// TwinCAT 3 PLC project ServoMotion_Library
// Title: ServoMotion_Lib
// Company: Chua Siang Poh
// Author: Chua Siang Poh
// ProjectVersion: 1.0
// Description: For projects that require at least 1 motion axis. The library is meant as an easy-to-setup module. Only requring the change of a parameter. Other motion functions are exposed as a method. Includes a very simple/crude type of linear interpolation.
// ProgramVersion: 3.1.0.8
// libraries:
//   Tc2_MC2, * (Beckhoff Automation GmbH)
//   Tc2_Standard, * (Beckhoff Automation GmbH)
//   Tc2_System, * (Beckhoff Automation GmbH)
//   Tc3_Interfaces, * (Beckhoff Automation GmbH)
//   Tc3_Module, * (Beckhoff Automation GmbH)
// project tree:
//   Custom Datatypes/ Motion_Axis.TcDUT, Motion_AxisGroup.TcDUT, Motion_HmiToPlc.TcDUT, Motion_PlcToHmi.TcDUT, ServoMotion_FunctionResult.TcDUT
//   GVL/ ServoMotion_GVL.TcGVL
//   / Interpolate.TcPOU, Servo.TcPOU, ServoMotion_Parameters.TcGVL
//   Version/ Global_Version.TcGVL
// (motion and I/O tree: see PLC project serialcommunication)
// real-time tasks:
//   TASK PlcTask: cycle T#10ms, priority 20, ADS port 350

// ---- Custom Datatypes/Motion_Axis.TcDUT
TYPE Motion_Axis :
STRUCT
	AXIS 					: AXIS_REF;
	HOME_CALIBRATION AT %I* : BOOL;
END_STRUCT
END_TYPE

// ---- Custom Datatypes/Motion_AxisGroup.TcDUT
TYPE Motion_AxisGroup :
STRUCT
	V_X			: LREAL;
	V_Y			: LREAL;
	X_AXIS		: INT;
	Y_AXIS		: INT;
	STATE		: INT;
	Y_IS_MASTER	: BOOL;
	X_DONE		: BOOL;
	Y_DONE		: BOOL;
END_STRUCT
END_TYPE

// ---- Custom Datatypes/Motion_HmiToPlc.TcDUT
TYPE Motion_HmiToPlc :
STRUCT
	TARGET_POSITION 	: LREAL;
	TARGET_VELOCITY 	: LREAL;
	TARGET_ACCELERATION : LREAL;
	TARGET_DECELERATION	: LREAL;
	TARGET_JERK			: LREAL;
	CONTROLLER_OVERRIDE	: LREAL;
	SERVO_ON			: BOOL;
	SERVO_ON_FW			: BOOL;
	SERVO_ON_BW			: BOOL;
	SERVO_OFF			: BOOL;
	SERVO_MOVE_ABS		: BOOL;
	SERVO_MOVE_REL		: BOOL;
	SERVO_HOME			: BOOL;
	SERVO_RESET			: BOOL;
	SERVO_JOG_MODE		: BOOL := FALSE;
	SERVO_JOG_FW_FAST	: BOOL;
	SERVO_JOG_BW_FAST	: BOOL;
	SERVO_JOG_FW_SLOW	: BOOL;
	SERVO_JOG_BW_SLOW	: BOOL;
END_STRUCT
END_TYPE

// ---- Custom Datatypes/Motion_PlcToHmi.TcDUT
TYPE Motion_PlcToHmi :
STRUCT
	actPos				: LREAL;
	actVelo				: LREAL;
	setPos				: LREAL; 
	setVelo 			: LREAL; 
	controller_override : LREAL;
	ErrorID				: UDINT;
	hasError			: BOOL;
	isDisabled 			: BOOL;
	isFwDisabled 		: BOOL;
	isBwDisabled 		: BOOL;
	isCalibrated		: BOOL;
	hasJob				: BOOL;
	isNotMoving 		: BOOL;
	isPositiveDirection : BOOL;
	isNegativeDirection : BOOL;            
    isInTarget 			: BOOL;            
    isInRange 			: BOOL;              
END_STRUCT
END_TYPE

// ---- Custom Datatypes/ServoMotion_FunctionResult.TcDUT
TYPE ServoMotion_FunctionResult :
(
	MOTION_OK := -1,
	MOTION_BUSY := 0,
	MOTION_UNKNOWN_AXIS,
	MOTION_UNKNOWN_AXIS_GROUP,
	MOTION_UNKNOWN_SAME_AXIS_IN_GROUP,
	MOTION_COMMAND_ABORTED,
	MOTION_ERROR
);
END_TYPE

// ---- GVL/ServoMotion_GVL.TcGVL
VAR_GLOBAL
	HmiToPlc	: ARRAY[1..MAX_AXES] OF Motion_HmiToPlc;
	PlcToHmi	: ARRAY[1..MAX_AXES] OF Motion_PlcToHmi;
	AXIS		: ARRAY[1..MAX_AXES] OF Motion_Axis;
END_VAR

// ---- ServoMotion_Parameters.TcGVL
VAR_GLOBAL CONSTANT
	MAX_AXES 		: INT := 2;
	MAX_AXIS_GROUPS	: INT := 1;
END_VAR

// ---- Version/Global_Version.TcGVL
// This function has been automatically generated from the project information.
VAR_GLOBAL CONSTANT
	{attribute 'const_non_replaced'}
	stLibVersion_ServoMotion_Lib : ST_LibVersion := (iMajor := 1, iMinor := 0, iBuild := 0, iRevision := 0, sVersion := '1.0');
END_VAR

// ---- Interpolate.TcPOU
FUNCTION_BLOCK Interpolate EXTENDS Servo
VAR_INPUT
END_VAR
VAR_OUTPUT
END_VAR
VAR
	fbGearIn 	: ARRAY [1..MAX_AXIS_GROUPS] OF MC_GEARIN;
	fbGearOut 	: ARRAY [1..MAX_AXIS_GROUPS] OF MC_GEAROUT;
	AXISGROUP	: ARRAY [1..MAX_AXIS_GROUPS] OF Motion_AxisGroup;
END_VAR

;

METHOD PUBLIC Set_AxisGroup : ServoMotion_FunctionResult
VAR_INPUT
	AXIS_GROUP_INDEX	: INT;
	X_AXIS_INDEX		: INT;
	Y_AXIS_INDEX		: INT;
END_VAR
IF AXIS_GROUP_INDEX < 1 OR AXIS_GROUP_INDEX > MAX_AXIS_GROUPS THEN
	Set_AxisGroup := ServoMotion_FunctionResult.MOTION_UNKNOWN_AXIS_GROUP;
ELSIF X_AXIS_INDEX < 1 OR X_AXIS_INDEX > MAX_AXES THEN
	Set_AxisGroup := ServoMotion_FunctionResult.MOTION_UNKNOWN_AXIS;
ELSIF Y_AXIS_INDEX < 1 OR Y_AXIS_INDEX > MAX_AXES THEN
	Set_AxisGroup := ServoMotion_FunctionResult.MOTION_UNKNOWN_AXIS;
ELSIF X_AXIS_INDEX = Y_AXIS_INDEX THEN
	Set_AxisGroup := ServoMotion_FunctionResult.MOTION_UNKNOWN_SAME_AXIS_IN_GROUP;
ELSE
	AXISGROUP[AXIS_GROUP_INDEX].X_AXIS := X_AXIS_INDEX;
	AXISGROUP[AXIS_GROUP_INDEX].Y_AXIS := Y_AXIS_INDEX;
	AXISGROUP[AXIS_GROUP_INDEX].STATE := -10;
	Set_AxisGroup := ServoMotion_FunctionResult.MOTION_OK;
END_IF
END_METHOD

METHOD PROTECTED Servo_GearIn : ServoMotion_FunctionResult
VAR_INPUT
	GROUP		: INT;
	MASTER		: INT;
	SLAVE		: INT;
	RATIO		: LREAL;
END_VAR
IF GROUP < 1 OR GROUP > MAX_AXIS_GROUPS THEN
	Servo_GearIn := ServoMotion_FunctionResult.MOTION_UNKNOWN_AXIS_GROUP;
ELSIF MASTER < 1 OR MASTER > MAX_AXES THEN
	Servo_GearIn := ServoMotion_FunctionResult.MOTION_UNKNOWN_AXIS;
ELSIF SLAVE < 1 OR SLAVE > MAX_AXES THEN
	Servo_GearIn := ServoMotion_FunctionResult.MOTION_UNKNOWN_AXIS;
ELSIF MASTER = SLAVE THEN
	Servo_GearIn := ServoMotion_FunctionResult.MOTION_UNKNOWN_SAME_AXIS_IN_GROUP;
ELSE
	fbGearIn[GROUP](
		Master:= AXIS[MASTER].AXIS, 
		Slave:= AXIS[SLAVE].AXIS, 
		Execute:= TRUE, 
		RatioNumerator:= RATIO, 
		RatioDenominator:= 1 );
	IF fbGearIn[GROUP].InGear THEN
		fbGearIn[GROUP](
			Master:= AXIS[MASTER].AXIS, 
			Slave:= AXIS[SLAVE].AXIS, 
			Execute:= FALSE );
		Servo_GearIn := ServoMotion_FunctionResult.MOTION_OK;
	ELSIF fbGearIn[GROUP].Error THEN
		fbGearIn[GROUP](
			Master:= AXIS[MASTER].AXIS, 
			Slave:= AXIS[SLAVE].AXIS, 
			Execute:= FALSE );
		Servo_GearIn := ServoMotion_FunctionResult.MOTION_ERROR;
	ELSIF fbGearIn[GROUP].CommandAborted THEN 
		fbGearIn[GROUP](
			Master:= AXIS[MASTER].AXIS, 
			Slave:= AXIS[SLAVE].AXIS, 
			Execute:= FALSE );
		Servo_GearIn := ServoMotion_FunctionResult.MOTION_COMMAND_ABORTED; 
	ELSE
		Servo_GearIn:= ServoMotion_FunctionResult.MOTION_BUSY;
	END_IF
END_IF
END_METHOD

METHOD PROTECTED Interpolate : ServoMotion_FunctionResult
VAR_INPUT
	GROUP			: INT;
	TO_X_POSITION	: LREAL;
	TO_Y_POSITION	: LREAL;
	VELOCITY		: LREAL;
END_VAR
VAR
	delta_t : LREAL;
	delta_x : LREAL;
	delta_y : LREAL;
	distance: LREAL;
END_VAR
IF GROUP < 1 OR GROUP > MAX_AXIS_GROUPS THEN
	Interpolate := ServoMotion_FunctionResult.MOTION_UNKNOWN_AXIS_GROUP;
ELSIF AXISGROUP[GROUP].X_AXIS < 1 OR AXISGROUP[GROUP].X_AXIS > MAX_AXES THEN
	Interpolate := ServoMotion_FunctionResult.MOTION_UNKNOWN_AXIS;
ELSIF AXISGROUP[GROUP].Y_AXIS < 1 OR AXISGROUP[GROUP].Y_AXIS > MAX_AXES THEN
	Interpolate := ServoMotion_FunctionResult.MOTION_UNKNOWN_AXIS;
ELSIF AXISGROUP[GROUP].X_AXIS = AXISGROUP[GROUP].Y_AXIS THEN
	Interpolate := ServoMotion_FunctionResult.MOTION_UNKNOWN_SAME_AXIS_IN_GROUP;
//ELSIF AXISGROUP[GROUP].STATE <> -10 THEN
//	Interpolate := ServoMotion_FunctionResult.MOTION_ERROR;
ELSE
 	CASE AXISGROUP[GROUP].STATE OF
	-10:
		delta_x := TO_X_POSITION - AXIS[AXISGROUP[GROUP].X_AXIS].AXIS.NcToPlc.ActPos;
		delta_y := TO_Y_POSITION - AXIS[AXISGROUP[GROUP].Y_AXIS].AXIS.NcToPlc.ActPos;
		distance:= SQRT((delta_x*delta_x) + (delta_y*delta_y));
		delta_t := distance/VELOCITY;
		AXISGROUP[GROUP].V_X := delta_x/delta_t;
		AXISGROUP[GROUP].V_Y := delta_y/delta_t;
		IF AXISGROUP[GROUP].V_X < 0.00001 AND AXISGROUP[GROUP].V_Y > 0.00001 THEN
			AXISGROUP[GROUP].Y_IS_MASTER := TRUE;
		ELSE
			AXISGROUP[GROUP].Y_IS_MASTER := FALSE;
		END_IF
		AXISGROUP[GROUP].STATE := 10;
		Interpolate := ServoMotion_FunctionResult.MOTION_BUSY;
	10:
		IF AXISGROUP[GROUP].Y_IS_MASTER THEN
			IF Servo_GearIn(GROUP,AXISGROUP[GROUP].Y_AXIS,AXISGROUP[GROUP].X_AXIS,AXISGROUP[GROUP].V_X/AXISGROUP[GROUP].V_Y) = ServoMotion_FunctionResult.MOTION_OK THEN
				AXISGROUP[GROUP].STATE := 20;
			END_IF
		ELSE
			IF Servo_GearIn(GROUP,AXISGROUP[GROUP].X_AXIS,AXISGROUP[GROUP].Y_AXIS,AXISGROUP[GROUP].V_Y/AXISGROUP[GROUP].V_X) = ServoMotion_FunctionResult.MOTION_OK THEN
				AXISGROUP[GROUP].STATE := 20;
			END_IF
		END_IF
		Interpolate := ServoMotion_FunctionResult.MOTION_BUSY;
	20: 
		IF AXISGROUP[GROUP].Y_IS_MASTER THEN
			IF Servo_MoveToPosition(AXISGROUP[GROUP].Y_AXIS, TO_Y_POSITION,ABS(AXISGROUP[GROUP].V_Y),0,0,0) = ServoMotion_FunctionResult.MOTION_OK THEN
				AXISGROUP[GROUP].STATE := 30;
			END_IF 
		ELSE
			IF Servo_MoveToPosition(AXISGROUP[GROUP].X_AXIS, TO_X_POSITION,ABS(AXISGROUP[GROUP].V_X),0,0,0) = ServoMotion_FunctionResult.MOTION_OK THEN
				AXISGROUP[GROUP].STATE := 30;
			END_IF
		END_IF
		Interpolate := ServoMotion_FunctionResult.MOTION_BUSY;
	30:
		IF AXISGROUP[GROUP].Y_IS_MASTER THEN
			fbGearOut[GROUP](
				Slave:= AXIS[AXISGROUP[GROUP].X_AXIS].AXIS, 
				Execute:= TRUE );
			IF fbGearOut[GROUP].Done THEN
				fbGearOut[GROUP](
					Slave:= AXIS[AXISGROUP[GROUP].X_AXIS].AXIS, 
					Execute:= FALSE );
				AXISGROUP[GROUP].STATE := -10;
				Interpolate := ServoMotion_FunctionResult.MOTION_OK;
			ELSIF fbGearOut[GROUP].Error THEN
				fbGearOut[GROUP](
					Slave:= AXIS[AXISGROUP[GROUP].X_AXIS].AXIS, 
					Execute:= FALSE );
				AXISGROUP[GROUP].STATE := -10;
				Interpolate := ServoMotion_FunctionResult.MOTION_ERROR;
			END_IF
		ELSE
			fbGearOut[GROUP](
				Slave:= AXIS[AXISGROUP[GROUP].Y_AXIS].AXIS, 
				Execute:= TRUE );
			IF fbGearOut[GROUP].Done THEN
				fbGearOut[GROUP](
					Slave:= AXIS[AXISGROUP[GROUP].Y_AXIS].AXIS, 
					Execute:= FALSE );
				AXISGROUP[GROUP].STATE := -10;
				Interpolate := ServoMotion_FunctionResult.MOTION_OK;
			ELSIF fbGearOut[GROUP].Error THEN
				fbGearOut[GROUP](
					Slave:= AXIS[AXISGROUP[GROUP].Y_AXIS].AXIS, 
					Execute:= FALSE );
				AXISGROUP[GROUP].STATE := -10;
				Interpolate := ServoMotion_FunctionResult.MOTION_ERROR;
			END_IF
		END_IF
	END_CASE
END_IF
END_METHOD

METHOD PUBLIC LinearInterpolate : ServoMotion_FunctionResult
VAR_INPUT
	GROUP 			: INT;
	TO_X_POSITION 	: LREAL;
	TO_Y_POSITION 	: LREAL;
	VELOCITY		: LREAL;
END_VAR
VAR
	delta_x : LREAL;
	delta_y : LREAL;
	delta_t : LREAL;
	distance: LREAL;
END_VAR
IF GROUP < 1 OR GROUP > MAX_AXIS_GROUPS THEN
	LinearInterpolate := ServoMotion_FunctionResult.MOTION_UNKNOWN_AXIS_GROUP;
ELSIF AXISGROUP[GROUP].X_AXIS < 1 OR AXISGROUP[GROUP].X_AXIS > MAX_AXES THEN
	LinearInterpolate := ServoMotion_FunctionResult.MOTION_UNKNOWN_AXIS;
ELSIF AXISGROUP[GROUP].Y_AXIS < 1 OR AXISGROUP[GROUP].Y_AXIS > MAX_AXES THEN
	LinearInterpolate := ServoMotion_FunctionResult.MOTION_UNKNOWN_AXIS;
ELSIF AXISGROUP[GROUP].X_AXIS = AXISGROUP[GROUP].Y_AXIS THEN
	LinearInterpolate := ServoMotion_FunctionResult.MOTION_UNKNOWN_SAME_AXIS_IN_GROUP;
ELSE
	CASE AXISGROUP[GROUP].STATE OF
	-10:
		delta_x := TO_X_POSITION - AXIS[AXISGROUP[GROUP].X_AXIS].AXIS.NcToPlc.ActPos;
		delta_y := TO_Y_POSITION - AXIS[AXISGROUP[GROUP].Y_AXIS].AXIS.NcToPlc.ActPos;
		distance:= SQRT((delta_x*delta_x) + (delta_y*delta_y));
		delta_t := distance/VELOCITY;
		AXISGROUP[GROUP].V_X := delta_x/delta_t;
		AXISGROUP[GROUP].V_Y := delta_y/delta_t;
		AXISGROUP[GROUP].STATE := 10;
		AXISGROUP[GROUP].X_DONE := FALSE;
		AXISGROUP[GROUP].Y_DONE := FALSE;
		LinearInterpolate := ServoMotion_FunctionResult.MOTION_BUSY;
		
	10:
		IF NOT AXISGROUP[GROUP].X_DONE THEN 
			IF Servo_MoveToPosition(AXISGROUP[GROUP].X_AXIS,TO_X_POSITION,ABS(AXISGROUP[GROUP].V_X),0,0,0) = ServoMotion_FunctionResult.MOTION_OK THEN 
				AXISGROUP[GROUP].X_DONE := TRUE;
			END_IF
		END_IF
		IF NOT AXISGROUP[GROUP].Y_DONE THEN 
			IF Servo_MoveToPosition(AXISGROUP[GROUP].Y_AXIS,TO_Y_POSITION,ABS(AXISGROUP[GROUP].V_Y),0,0,0) = ServoMotion_FunctionResult.MOTION_OK THEN
				AXISGROUP[GROUP].Y_DONE := TRUE;
			END_IF
		END_IF
		IF AXISGROUP[GROUP].X_DONE AND AXISGROUP[GROUP].Y_DONE THEN
			AXISGROUP[GROUP].STATE := 20;
		ELSE
			LinearInterpolate := ServoMotion_FunctionResult.MOTION_BUSY;
		END_IF
	20:
		AXISGROUP[GROUP].STATE := -10;
		AXISGROUP[GROUP].X_DONE := FALSE;
		AXISGROUP[GROUP].Y_DONE := FALSE;
		LinearInterpolate := ServoMotion_FunctionResult.MOTION_OK;
	END_CASE
END_IF
END_METHOD

END_FUNCTION_BLOCK

// ---- Servo.TcPOU
FUNCTION_BLOCK Servo
VAR_INPUT
	HMI_MODE : BOOL;
END_VAR
VAR_OUTPUT
END_VAR
VAR
	fbPower 	: ARRAY [1..MAX_AXES] OF MC_POWER;
	fbReset 	: ARRAY [1..MAX_AXES] OF MC_RESET;
	fbHome		: ARRAY	[1..MAX_AXES] OF MC_HOME;
	fbMoveA 	: ARRAY [1..MAX_AXES] OF MC_MOVEABSOLUTE;
	fbMoveR 	: ARRAY [1..MAX_AXES] OF MC_MOVERELATIVE;
	fbJog		: ARRAY [1..MAX_AXES] OF MC_JOG;
	fbHalt	 	: ARRAY [1..MAX_AXES] OF MC_HALT;
	i			: INT;
END_VAR

IF HMI_MODE THEN 
	FOR i := 1 TO MAX_AXES BY 1 DO
		ACT_UpdateStatus();
		IF HmiToPlc[i].SERVO_OFF THEN
			ACT_Off();
		ELSIF HmiToPlc[i].SERVO_ON THEN 
			ACT_On();
		END_IF
		IF NOT HmiToPlc[i].SERVO_JOG_MODE THEN 
			Servo_Jog_Stop(i);
			IF HmiToPlc[i].SERVO_MOVE_ABS THEN
				ACT_MoveToPosition();
			END_IF
			IF HmiToPlc[i].SERVO_MOVE_REL THEN
				ACT_MoveByDistance();
			END_IF
		ELSE
			ACT_Jog();
		END_IF
	END_FOR
END_IF

ACTION ACT_On:
Servo_On(i, HmiToPlc[i].SERVO_ON_FW, HmiToPlc[i].SERVO_ON_BW, HmiToPlc[i].CONTROLLER_OVERRIDE);
END_ACTION

METHOD PUBLIC Servo_Home : ServoMotion_FunctionResult
VAR_INPUT
	INDEX : INT;
END_VAR
IF INDEX > MAX_AXES OR INDEX < 1 THEN 
	Servo_Home := ServoMotion_FunctionResult.MOTION_UNKNOWN_AXIS;
ELSE
	fbHome[INDEX](
		Axis:= AXIS[INDEX].AXIS, 
		Execute:= TRUE, 
		Position:= 0, 
		HomingMode:= MC_DefaultHoming, 
		bCalibrationCam:= AXIS[INDEX].HOME_CALIBRATION );
	IF fbHome[INDEX].Error THEN
		fbHome[INDEX](
			Axis:= AXIS[INDEX].AXIS, 
			Execute:= FALSE );
		Servo_Home := ServoMotion_FunctionResult.MOTION_ERROR;
	ELSIF fbHome[INDEX].CommandAborted THEN
		fbHome[INDEX](
			Axis:= AXIS[INDEX].AXIS, 
			Execute:= FALSE );
		Servo_Home := ServoMotion_FunctionResult.MOTION_COMMAND_ABORTED;
	ELSIF fbHome[INDEX].Done THEN
		fbHome[INDEX](
			Axis:= AXIS[INDEX].AXIS, 
			Execute:= FALSE );
		Servo_Home := ServoMotion_FunctionResult.MOTION_OK;
	ELSE
		Servo_Home := ServoMotion_FunctionResult.MOTION_BUSY;
	END_IF
END_IF
END_METHOD

METHOD PUBLIC Servo_Jog_Stop : ServoMotion_FunctionResult
VAR_INPUT
	INDEX : INT;
END_VAR
fbJog[INDEX](
	Axis:= AXIS[INDEX].AXIS, 
	JogForward:= FALSE, 
	JogBackwards:= FALSE );
IF fbJog[INDEX].Error THEN 
	Servo_Jog_Stop := ServoMotion_FunctionResult.MOTION_ERROR;
ELSE
	Servo_Jog_Stop := ServoMotion_FunctionResult.MOTION_OK;
END_IF
END_METHOD

METHOD PUBLIC Servo_Off : ServoMotion_FunctionResult
VAR_INPUT
	INDEX : INT;
END_VAR
IF INDEX > MAX_AXES OR INDEX < 1 THEN 
	Servo_Off := ServoMotion_FunctionResult.MOTION_UNKNOWN_AXIS;
ELSE
	fbPower[INDEX](
		Axis:= AXIS[INDEX].AXIS, 
		Enable:= FALSE, 
		Enable_Positive:= FALSE, 
		Enable_Negative:= FALSE, 
		Override:= 0 );
	IF fbPower[INDEX].Error THEN
		Servo_Off := ServoMotion_FunctionResult.MOTION_ERROR;
	ELSIF NOT fbPower[INDEX].Status THEN
		Servo_Off := ServoMotion_FunctionResult.MOTION_OK;
	ELSE
		Servo_Off := ServoMotion_FunctionResult.MOTION_BUSY;
	END_IF
END_IF
END_METHOD

ACTION ACT_MoveToPosition:
CASE Servo_MoveToPosition(i,HmiToPlc[i].TARGET_POSITION,HmiToPlc[i].TARGET_VELOCITY,HmiToPlc[i].TARGET_ACCELERATION,HmiToPlc[i].TARGET_DECELERATION,HmiToPlc[i].TARGET_JERK) OF
ServoMotion_FunctionResult.MOTION_UNKNOWN_AXIS:
	;
ServoMotion_FunctionResult.MOTION_COMMAND_ABORTED: 
	;
ServoMotion_FunctionResult.MOTION_ERROR:
	;
ServoMotion_FunctionResult.MOTION_BUSY: 
	;
ServoMotion_FunctionResult.MOTION_OK:
	;
END_CASE
END_ACTION

PROPERTY PUBLIC AXIS_COUNT : INT
GET
AXIS_COUNT := MAX_AXES;
END_GET
END_PROPERTY

METHOD PUBLIC Servo_MoveToPosition : ServoMotion_FunctionResult
VAR_INPUT
	INDEX 			: INT;
	POSITION		: LREAL;
	VELOCITY		: LREAL;
	ACCELERATION	: LREAL;
	DECELERATION	: LREAL;
	JERK			: LREAL;
END_VAR
IF INDEX > MAX_AXES OR INDEX < 1 AND VELOCITY <= 0 THEN 
	Servo_MoveToPosition := ServoMotion_FunctionResult.MOTION_UNKNOWN_AXIS;
ELSE
	fbMoveA[INDEX](
		Axis:= AXIS[INDEX].AXIS, 
		Execute:= TRUE, 
		Position:= POSITION, 
		Velocity:= VELOCITY, 
		Acceleration:= ACCELERATION, 
		Deceleration:= DECELERATION, 
		Jerk:= JERK );
	IF fbMoveA[INDEX].Error THEN
		fbMoveA[INDEX](
			Axis:= AXIS[INDEX].AXIS, 
			Execute:= FALSE );
		Servo_MoveToPosition := ServoMotion_FunctionResult.MOTION_ERROR;
	ELSIF fbMoveA[INDEX].CommandAborted THEN
		fbMoveA[INDEX](
			Axis:= AXIS[INDEX].AXIS, 
			Execute:= FALSE );
		Servo_MoveToPosition := ServoMotion_FunctionResult.MOTION_COMMAND_ABORTED;
	ELSIF fbMoveA[INDEX].Done THEN
		fbMoveA[INDEX](
			Axis:= AXIS[INDEX].AXIS, 
			Execute:= FALSE );
		Servo_MoveToPosition := ServoMotion_FunctionResult.MOTION_OK;
	ELSE
		Servo_MoveToPosition := ServoMotion_FunctionResult.MOTION_BUSY;
	END_IF
END_IF
END_METHOD

ACTION ACT_Off:
Servo_Off(i);
END_ACTION

METHOD PUBLIC Servo_Halt : ServoMotion_FunctionResult
VAR_INPUT
	INDEX : INT;
END_VAR
IF INDEX > MAX_AXES OR INDEX < 1 THEN 
	Servo_Halt := ServoMotion_FunctionResult.MOTION_UNKNOWN_AXIS;
ELSE
	fbHalt[INDEX](
		Axis:= AXIS[INDEX].AXIS, 
		Execute:= TRUE );
	fbMoveA[INDEX](
		Axis:= AXIS[INDEX].AXIS, 
		Execute:= FALSE );
	fbMoveR[INDEX](
		Axis:= AXIS[INDEX].AXIS, 
		Execute:= FALSE );
	IF fbHalt[INDEX].Error THEN
		fbHalt[INDEX](
			Axis:= AXIS[INDEX].AXIS, 
			Execute:= FALSE );
		Servo_Halt := ServoMotion_FunctionResult.MOTION_ERROR;
	ELSIF fbHalt[INDEX].CommandAborted THEN
		fbHalt[INDEX](
			Axis:= AXIS[INDEX].AXIS, 
			Execute:= FALSE );
		Servo_Halt := ServoMotion_FunctionResult.MOTION_COMMAND_ABORTED;
	ELSIF fbHalt[INDEX].Done THEN
		fbHalt[INDEX](
			Axis:= AXIS[INDEX].AXIS, 
			Execute:= FALSE );
		Servo_Halt := ServoMotion_FunctionResult.MOTION_OK;
	ELSE
		Servo_Halt := ServoMotion_FunctionResult.MOTION_BUSY;
	END_IF
END_IF
END_METHOD

ACTION ACT_MoveByDistance:
CASE Servo_MoveByDistance(i,HmiToPlc[i].TARGET_POSITION,HmiToPlc[i].TARGET_VELOCITY,HmiToPlc[i].TARGET_ACCELERATION,HmiToPlc[i].TARGET_DECELERATION,HmiToPlc[i].TARGET_JERK) OF
ServoMotion_FunctionResult.MOTION_UNKNOWN_AXIS:
	;
ServoMotion_FunctionResult.MOTION_COMMAND_ABORTED: 
	;
ServoMotion_FunctionResult.MOTION_ERROR:
	;
ServoMotion_FunctionResult.MOTION_BUSY: 
	;
ServoMotion_FunctionResult.MOTION_OK:
	;
END_CASE
END_ACTION

METHOD PUBLIC Servo_Jog_Start : ServoMotion_FunctionResult
VAR_INPUT
	INDEX		: INT;
	REVERSE		: BOOL := FALSE;
	FAST_MODE	: BOOL := FALSE;
END_VAR
IF FAST_MODE THEN 
	fbJog[INDEX].Mode := MC_JOGMODE_STANDARD_FAST;
ELSE
	fbJog[INDEX].Mode := MC_JOGMODE_STANDARD_SLOW;
END_IF

fbJog[INDEX](
	Axis:= AXIS[INDEX].AXIS, 
	JogForward:= NOT REVERSE, 
	JogBackwards:= REVERSE );
IF fbJog[INDEX].Error THEN 
	Servo_Jog_Start := ServoMotion_FunctionResult.MOTION_ERROR;
ELSIF AXIS[INDEX].AXIS.Status.Moving THEN 
	Servo_Jog_Start := ServoMotion_FunctionResult.MOTION_OK;
END_IF
END_METHOD

PROPERTY AxisGroup_Count : INT
GET
AXISGROUP_Count := MAX_AXIS_GROUPS;
END_GET
END_PROPERTY

ACTION ACT_Reset:
IF Servo_Reset(i) = ServoMotion_FunctionResult.MOTION_OK THEN
	HmiToPlc[i].SERVO_RESET := FALSE;
END_IF
END_ACTION

METHOD PUBLIC Servo_MoveByDistance : ServoMotion_FunctionResult
VAR_INPUT
	INDEX 			: INT;
	DISTANCE 		: LREAL;
	VELOCITY 		: LREAL;
	ACCELERATION 	: LREAL;
	DECELERATION 	: LREAL;
	JERK 			: LREAL;
END_VAR
IF INDEX > MAX_AXES OR INDEX < 1 AND VELOCITY <= 0 THEN 
	Servo_MoveByDistance := ServoMotion_FunctionResult.MOTION_UNKNOWN_AXIS;
ELSE
	fbMoveR[INDEX](
		Axis:= AXIS[INDEX].AXIS, 
		Execute:= TRUE, 
		Distance:= DISTANCE, 
		Velocity:= VELOCITY, 
		Acceleration:= ACCELERATION, 
		Deceleration:= DECELERATION, 
		Jerk:= JERK );
	IF fbMoveR[INDEX].Error THEN
		fbMoveR[INDEX](
			Axis:= AXIS[INDEX].AXIS, 
			Execute:= FALSE );
		Servo_MoveByDistance := ServoMotion_FunctionResult.MOTION_ERROR;
	ELSIF fbMoveR[INDEX].CommandAborted THEN
		fbMoveR[INDEX](
			Axis:= AXIS[INDEX].AXIS, 
			Execute:= FALSE );
		Servo_MoveByDistance := ServoMotion_FunctionResult.MOTION_COMMAND_ABORTED;
	ELSIF fbMoveR[INDEX].Done THEN
		fbMoveR[INDEX](
			Axis:= AXIS[INDEX].AXIS, 
			Execute:= FALSE );
		Servo_MoveByDistance := ServoMotion_FunctionResult.MOTION_OK;
	ELSE
		Servo_MoveByDistance := ServoMotion_FunctionResult.MOTION_BUSY;
	END_IF
END_IF
END_METHOD

ACTION ACT_Jog:
IF HmiToPlc[i].SERVO_JOG_FW_FAST THEN
	Servo_Jog_Start(i, FALSE, TRUE);
ELSIF HmiToPlc[i].SERVO_JOG_FW_SLOW THEN
	Servo_Jog_Start(i, FALSE, FALSE);
ELSIF HmiToPlc[i].SERVO_JOG_BW_FAST THEN
	Servo_Jog_Start(i, TRUE, TRUE);
ELSIF HmiToPlc[i].SERVO_JOG_BW_SLOW THEN
	Servo_Jog_Start(i, TRUE, FALSE);
ELSE
	Servo_Jog_Stop(i);
END_IF
END_ACTION

METHOD Servo_On : ServoMotion_FunctionResult
VAR_INPUT
	INDEX : INT;
	ENABLE_FW 	: BOOL;
	ENABLE_BW	: BOOL;
	OVERRIDE	: LREAL;
END_VAR
IF INDEX > MAX_AXES OR INDEX < 1 THEN 
	Servo_On := ServoMotion_FunctionResult.MOTION_UNKNOWN_AXIS;
ELSE
	fbPower[INDEX](
		Axis:= AXIS[INDEX].AXIS, 
		Enable:= TRUE, 
		Enable_Positive:= ENABLE_FW, 
		Enable_Negative:= ENABLE_BW, 
		Override:= OVERRIDE );
	IF fbPower[INDEX].Error THEN
		Servo_On := ServoMotion_FunctionResult.MOTION_ERROR;
	ELSIF fbPower[INDEX].Status THEN
		Servo_On := ServoMotion_FunctionResult.MOTION_OK;
	ELSE
		Servo_On := ServoMotion_FunctionResult.MOTION_BUSY;
	END_IF
END_IF
END_METHOD

METHOD PUBLIC Servo_Reset : ServoMotion_FunctionResult
VAR_INPUT
	INDEX :INT;
END_VAR
IF INDEX > MAX_AXES OR INDEX < 1 THEN 
	Servo_Reset := ServoMotion_FunctionResult.MOTION_UNKNOWN_AXIS;
ELSE
	fbReset[INDEX](
		Axis:= AXIS[INDEX].AXIS, 
		Execute:= TRUE );
	IF fbReset[INDEX].Error THEN
		fbReset[INDEX](
			Axis:= AXIS[INDEX].AXIS, 
			Execute:= FALSE );
		Servo_Reset := ServoMotion_FunctionResult.MOTION_ERROR;
	ELSIF fbReset[INDEX].Done THEN
		fbReset[INDEX](
			Axis:= AXIS[INDEX].AXIS, 
			Execute:= FALSE );
		Servo_Reset := ServoMotion_FunctionResult.MOTION_OK;
	ELSE
		Servo_Reset := ServoMotion_FunctionResult.MOTION_BUSY;
	END_IF
END_IF
END_METHOD

ACTION ACT_UpdateStatus:
AXIS[i].AXIS.ReadStatus();
PlcToHmi[i].actPos	:= AXIS[i].AXIS.NcToPlc.ActPos;
PlcToHmi[i].actVelo := AXIS[i].AXIS.NcToPlc.ActVelo;
PlcToHmi[i].setPos	:= AXIS[i].AXIS.NcToPlc.SetPos;
PlcToHmi[i].setVelo := AXIS[i].AXIS.NcToPlc.SetVelo;
PlcToHmi[i].controller_override := fbPower[i].Override;
PlcToHmi[i].hasError := AXIS[i].AXIS.Status.Error;
PlcToHmi[i].ErrorID := AXIS[i].AXIS.Status.ErrorID;
PlcToHmi[i].isBwDisabled := NOT fbPower[i].Enable_Negative;
PlcToHmi[i].isFwDisabled := NOT fbPower[i].Enable_Positive;
PlcToHmi[i].isCalibrated := AXIS[i].AXIS.Status.Homed;
PlcToHmi[i].isDisabled := AXIS[i].AXIS.Status.Disabled;
PlcToHmi[i].isInRange := AXIS[i].AXIS.Status.InPositionArea;
PlcToHmi[i].isInTarget := AXIS[i].AXIS.Status.InTargetPosition;
PlcToHmi[i].isNegativeDirection := AXIS[i].AXIS.Status.NegativeDirection;
PlcToHmi[i].isNotMoving := AXIS[i].AXIS.Status.NotMoving;
PlcToHmi[i].isPositiveDirection := AXIS[i].AXIS.Status.PositiveDirection;
END_ACTION

END_FUNCTION_BLOCK
